// SIMATIC S7-200 project (STEP 7-Micro/WIN), CPU 224XP REL 02.00

ORGANIZATION_BLOCK 主:OB1
TITLE=程序注解
BEGIN
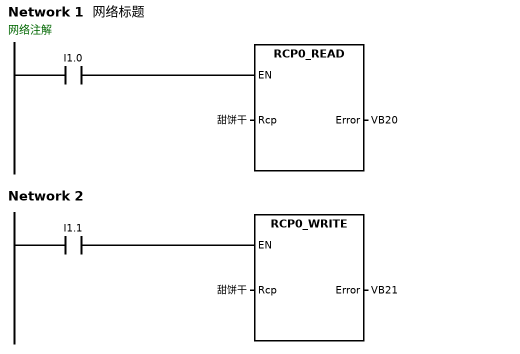
Network 1 // 网络标题
// 网络注解
LD     I1.0
CALL   RCP0_READ:SBR1, 甜饼干, VB20
Network 2
LD     I1.1
CALL   RCP0_WRITE:SBR2, 甜饼干, VB21
END_ORGANIZATION_BLOCK

// SBR1: protected block, not included

// SBR2: protected block, not included

// (further data pages could not be read)
